Universal Robots PolyScope program: program3.urp

Program program3 (installation=default directory=/ursim/programs createdIn=3.15.8.106339 lastSavedIn=3.15.8.106339 robotSerialNumber=2018359999)
Calibrated DH parameters: a=[0, -0.425, -0.39225, 0, 0, 0]; d=[0.089159, 0, 0, 0.10915, 0.09465, 0.0823]; alpha=[1.570796, 0, 0, 1.570796, -1.570796, 0]; deltaTheta=[0, 0, 0, 0, 0, 0]
Robot Program (runOnlyOnce=false)
  Script file /ursim/programs/programa3.script
    |   set_gravity([0.0, 0.0, 9.82])
    |   set_tcp(p[0.0,0.0,0.0,0.0,0.0,0.0])
    |   set_payload(2.0)
    |   set_tool_voltage(0)
    |   global v = 0.2
    |   global a = 0.5
    | 
    |   while (True):
    |     popup("Iniciando rutina Pick and Place", "Programa 3", False, False, True)
    | 
    |     movej(p[0.300, 0.000, 0.300, 3.14, 0.0, 0.0], a, v)
    | 
    |     movej(p[0.250, -0.100, 0.300, 3.14, 0.0, 0.0], a, v)
    |     movej(p[0.250, -0.100, 0.150, 3.14, 0.0, 0.0], a, v)
    |     set_digital_out(0, True)
    |     sleep(0.5)
    |     movej(p[0.250, -0.100, 0.250, 3.14, 0.0, 0.0], a, v)
    |     movej(p[0.350, 0.100, 0.250, 3.14, 0.0, 0.0], a, v)
    |     movej(p[0.350, 0.100, 0.150, 3.14, 0.0, 0.0], a, v)
    |     set_digital_out(0, False)
    |     sleep(0.5)
    |     movej(p[0.350, 0.100, 0.250, 3.14, 0.0, 0.0], a, v)
    | 
    |     movej(p[0.400, -0.100, 0.300, 3.14, 0.0, 0.0], a, v)
    |     movej(p[0.400, -0.100, 0.150, 3.14, 0.0, 0.0], a, v)
    |     set_digital_out(0, True)
    |     sleep(0.5)
    |     movej(p[0.400, -0.100, 0.250, 3.14, 0.0, 0.0], a, v)
    |     movej(p[0.450, 0.100, 0.250, 3.14, 0.0, 0.0], a, v)
    |     movej(p[0.450, 0.100, 0.150, 3.14, 0.0, 0.0], a, v)
    |     set_digital_out(0, False)
    |     sleep(0.5)
    |     movej(p[0.450, 0.100, 0.250, 3.14, 0.0, 0.0], a, v)
    | 
    |     movej(p[0.300, 0.000, 0.300, 3.14, 0.0, 0.0], a, v)
    | 
    |     popup("Rutina completada. Active entrada digital DI[0] para reiniciar.", "Esperando confirmación", False, False, True)
    |     while (not get_digital_in(0)):
    |       sleep(0.1)
    |     end
    |   end
